Universal Robots PolyScope program: main.urp

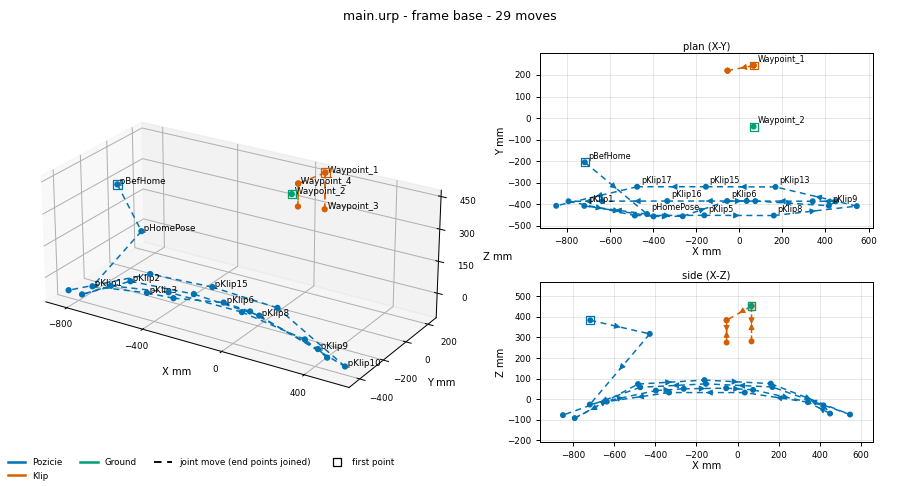
[picture p0: tool path of main.urp in frame base, 29 of 29 moves have a stored position in this frame; points joined in program order, loops and branches not executed]
Program main (installation=default directory=/programs/standart createdIn=5.9.4.1031232 lastSavedIn=3.15.3.106223 robotSerialNumber=2019351917)
Calibrated DH parameters: a=[0.000102, -0.047078, -0.0018, 0.000113, -0.000057, 0]; d=[0.089076, 134.205243, 65.197866, -199.293136, 0.094778, 0.082594]; alpha=[1.569561, -0.003151, -0.001967, 1.571153, -1.570968, 0]; deltaTheta=[0.00002, -1.459967, -0.106279, 1.566186, -0.000048, 0.000035]
Robot Program (runOnlyOnce=false)
  pTarget := p[0,0,0,0,0,0]
  nKlipNo := 1
  SuppressedNode
    bInHome := False
  Script file /programs/standart/loop.script
    | def main():
    | SetMovementsExtParams()
    | while (True):
    |     global niActionNo = read_input_integer_register(2)
    |     sync()
    | 	if (0 == niActionNo):
    | 		sync()
    | 	elif (1 == niActionNo):
    | 		if (read_output_integer_register(2)==255):
    |                                       Klip()
    | 	                  end
    | 	elif (100 == niActionNo):
    | 		if (read_output_integer_register(2)==255):
    | 		Ground()
    | 		end
    | 	elif (254 == niActionNo):
    | 		if (read_output_integer_register(2)==255):
    | 		SetMovementsExtParams ()
    | 		WriteMovementsExtParams ()
    | 		end
    | 	elif (255 == niActionNo):
    | 		sync()
    | 	else:
    | 		popup("nespravne cislo", "Message", False, True, blocking=False)
    | 		halt
    | 	end
    | 	global qActionNumber = niActionNo
    | 	WriteMovementsExtParams ()
    |                   sync()
    | end
    | end
    | def SetMovementsExtParams():
    |     global qActionNumber = read_input_integer_register(2)
    |     global ActGlobalSpeed=read_input_integer_register(3)
    |     global ActualToolNmbr=read_input_integer_register(4)
    |     global ActualWobjNmbr=read_input_integer_register(5)
    |     global ActualPointNmbr=read_input_integer_register(6)
    |     global ActUsrSpecSpd1=read_input_float_register(0)
    |     global ActUsrSpecSpd2=read_input_float_register(1)
    |     global ActCoordX=read_input_float_register(2)
    |     global ActCoordY=read_input_float_register(3)
    |     global ActCoordZ=read_input_float_register(4)
    |     global ActCoordRx=read_input_float_register(5)
    |     global ActCoordRy=read_input_float_register(6)
    |     global ActCoordRz=read_input_float_register(7)
    | end
    | def WriteMovementsExtParams():
    |     write_output_integer_register(2, qActionNumber)
    |     write_output_integer_register(3, ActGlobalSpeed)
    |     write_output_integer_register(4, ActualToolNmbr)
    |     write_output_integer_register(5, ActualWobjNmbr)
    |     write_output_integer_register(6, ActualPointNmbr)
    |     write_output_float_register(0, ActUsrSpecSpd1)
    |     write_output_float_register(1, ActUsrSpecSpd2)
    |     write_output_float_register(2, ActCoordX)
    |     write_output_float_register(3, ActCoordY)
    |     write_output_float_register(4, ActCoordZ)
    |     write_output_float_register(5, ActCoordRx)
    |     write_output_float_register(6, ActCoordRy)
    |     write_output_float_register(7, ActCoordRz)
    | end
  bTest := False
  SuppressedNode
    ipLastPos := get_actual_tcp_pose()
  SuppressedNode
    Call Ground
  Script: main()
SubProgram Pozicie (keepSynchronizedWithDisk=false)
  MoveJ speed 60 deg/s, acceleration 80 deg/s^2 (useActiveTCP=false) tcp=klipBezProtikus
    Waypoint pBefHome: TCP in base x=-715.649 y=-205.001 z=383.699 mm, rx=-2.2037 ry=-0.1236 rz=2.19 rad; joints [-138.345, -84.396, -124.639, -152.449, -62.006, -181.389] deg; flange x=-522.449 y=-193.771 z=341.759 mm, rx=-1.0723 ry=-1.4196 rz=1.3498 rad
    SuppressedNode
      Waypoint Waypoint_46: TCP in base x=-415.026 y=-230.779 z=167.281 mm, rx=-1.4886 ry=-2.6151 rz=0.3802 rad; joints [224.112, -91.25, -119.014, -236.004, -90.455, -253.965] deg; flange x=-396.865 y=-162.684 z=352.334 mm, rx=0.7585 ry=-2.9968 rz=0.0685 rad
    Waypoint pHomePose: motionParameters(blendRadius=0.05); TCP in base x=-426.741 y=-445.009 z=317.531 mm, rx=0.09 ry=-2.3315 rz=2.0367 rad; joints [-141.68, -91.952, -115.104, -182.866, -136.488, -294.8] deg; flange x=-471.084 y=-254.443 z=348.022 mm, rx=1.4686 ry=-1.4379 rz=0.9969 rad
  MoveJ speed 60 deg/s, acceleration 80 deg/s^2 (useActiveTCP=false) tcp=klipProtitlak
    Waypoint pKlip1: motionParameters(jointSpeed=2.094395 jointAcceleration=3.490659 cartesianSpeed=0.25 cartesianAcceleration=1.2); TCP in base x=-717.916 y=-407.007 z=-25.646 mm, rx=-2.1837 ry=2.0431 rz=-0.2819 rad; joints [-139.39, -122.492, -100.341, -46.423, -267.896, -230.294] deg; flange x=-758.162 y=-445.184 z=164.444 mm, rx=3.0989 ry=0.0292 rz=0.0301 rad
    Waypoint pKlip3: TCP in base x=-397.127 y=-455.596 z=42.237 mm, rx=-2.2464 ry=2.1402 rz=-0.0817 rad; joints [-116.855, -94.906, -132.082, -38.147, -277.33, -207.158] deg; flange x=-408.449 y=-427.485 z=238.512 mm, rx=3.1133 ry=0.0064 rz=-0.2302 rad
    Waypoint pKlip4: TCP in base x=-261.696 y=-455.216 z=50.966 mm, rx=-2.2467 ry=2.1402 rz=-0.0816 rad; joints [-102.622, -85.622, -139.646, -41.752, -278.247, -192.808] deg; flange x=-273.005 y=-427.094 z=247.24 mm, rx=3.1132 ry=0.0066 rz=-0.2303 rad
    Waypoint pKlip6: TCP in base x=-55.729 y=-384.407 z=53.915 mm, rx=2.2671 ry=-2.1584 rz=0.0011 rad; joints [-71.993, -75.789, -145.674, -51.415, -282.439, -161.677] deg; flange x=-50.779 y=-426.253 z=247.399 mm, rx=3.1035 ry=0.0081 rz=-0.3413 rad
    Waypoint pKlip7: TCP in base x=74.794 y=-384.809 z=45.787 mm, rx=2.2668 ry=-2.1583 rz=0.0012 rad; joints [-55.209, -77.405, -144.751, -54.17, -281.1, -144.583] deg; flange x=79.767 y=-426.6 z=239.281 mm, rx=3.1032 ry=0.008 rz=-0.3415 rad
    Waypoint pKlip9: TCP in base x=415.982 y=-406.314 z=-29.655 mm, rx=2.0484 ry=-1.9483 rz=-0.4078 rad; joints [-26.071, -109.42, -118.061, -74.534, -286.071, -111.582] deg; flange x=495.201 y=-447.711 z=147.042 mm, rx=2.9746 ry=0.0123 rz=-0.9451 rad
    SuppressedNode
      Waypoint Waypoint_36: TCP in base x=324.659 y=-377.766 z=383.702 mm, rx=-0.149 ry=1.7717 rz=-0.7957 rad; joints [322.849, -58.337, -129.745, -187.968, -109.913, 142.997] deg; flange x=158.512 y=-281.184 z=433.798 mm, rx=-1.7432 ry=1.3314 rz=-1.567 rad
    Waypoint pKlip11: TCP in base x=448.509 y=-385.741 z=-69.2 mm, rx=-2.1761 ry=-2.1899 rz=0.049 rad; joints [-21.41, -106.712, -137.424, -18.115, -266.245, 71.195] deg; flange x=458.564 y=-345.107 z=124.344 mm, rx=0.0574 ry=2.9899 rz=0.0308 rad
    Waypoint pKlip12: TCP in base x=341.02 y=-385.606 z=-13.953 mm, rx=-2.1522 ry=-2.1654 rz=0.1026 rad; joints [-25.586, -93.527, -143.331, -28.169, -266.914, 66.968] deg; flange x=360.406 y=-344.605 z=178.802 mm, rx=0.0584 ry=3.0382 rz=0.027 rad
    Waypoint pKlip14: TCP in base x=34.614 y=-384.474 z=32.579 mm, rx=-2.1881 ry=-2.2026 rz=0.0261 rad; joints [-58.228, -68.011, -154.767, -42.655, -261.175, 34.579] deg; flange x=40.264 y=-343.538 z=226.238 mm, rx=0.0562 ry=2.9672 rz=0.029 rad
    Waypoint pKlip16: TCP in base x=-333.423 y=-384.697 z=32.621 mm, rx=-2.1593 ry=-2.2797 rz=-0.0282 rad; joints [-117.379, -86.002, -139.546, -51.671, -259.578, -28.311] deg; flange x=-339.362 y=-343.904 z=226.302 mm, rx=-0.0144 ry=2.9183 rz=0.037 rad
    Waypoint pKlip18: TCP in base x=-635.307 y=-385.022 z=-11.351 mm, rx=2.0897 ry=2.2082 rz=0.1692 rad; joints [-141.865, -112.773, -110.469, -63.994, -259.039, -53.917] deg; flange x=-667.328 y=-344.256 z=179.762 mm, rx=-0.0161 ry=2.7829 rz=0.0348 rad
    Waypoint pKlip19: TCP in base x=-791.11 y=-385.677 z=-91.337 mm, rx=2.0027 ry=2.1167 rz=0.3408 rad; joints [-149.226, -131.492, -87.605, -78.107, -257.456, -62.68] deg; flange x=-853.946 y=-347.011 z=92.424 mm, rx=-0.0152 ry=2.6186 rz=0.0469 rad
  MoveJ speed 60 deg/s, acceleration 80 deg/s^2 (useActiveTCP=false) tcp=klipBezProtikus
    Waypoint pKlip2: TCP in base x=-483.859 y=-451.884 z=73.894 mm, rx=-2.2466 ry=2.1403 rz=-0.0817 rad; joints [-120.808, -101.736, -119.856, -43.059, -277.036, -211.134] deg; flange x=-492.737 y=-493.65 z=267.254 mm, rx=3.1132 ry=0.0065 rz=-0.2303 rad
    Waypoint pKlip5: TCP in base x=-161.364 y=-450.889 z=93.263 mm, rx=2.2668 ry=-2.1584 rz=0.0013 rad; joints [-87.222, -82.787, -136.209, -50.492, -282.819, -177.268] deg; flange x=-156.42 y=-492.687 z=286.757 mm, rx=3.1033 ry=0.0079 rz=-0.3413 rad
    Waypoint pKlip8: TCP in base x=160.789 y=-451.854 z=75.97 mm, rx=2.2666 ry=-2.1584 rz=0.0036 rad; joints [-51.599, -84.791, -134.791, -57.341, -280.729, -140.913] deg; flange x=165.557 y=-493.433 z=269.515 mm, rx=3.1023 ry=0.0076 rz=-0.3398 rad
    Waypoint pKlip10: TCP in base x=545.477 y=-408.071 z=-73.997 mm, rx=-0.0027 ry=-3.1325 rz=-0.0126 rad; joints [-26.569, -110.661, -126.204, -39.275, -259.338, -24.326] deg; flange x=503.576 y=-410.94 z=119.516 mm, rx=-2.0629 ry=2.1594 rz=0.2484 rad
    Waypoint pKlip13: TCP in base x=168.592 y=-319.265 z=59.545 mm, rx=-2.1886 ry=-2.2026 rz=0.0269 rad; joints [-30.415, -60.616, -155.192, -45.97, -264.32, 62.469] deg; flange x=174.28 y=-278.219 z=253.179 mm, rx=0.0565 ry=2.9673 rz=0.0281 rad
    Waypoint pKlip15: TCP in base x=-154.177 y=-318.207 z=74.988 mm, rx=-2.1599 ry=-2.2798 rz=-0.0278 rad; joints [-93.971, -58.689, -151.594, -62.02, -257.408, -4.458] deg; flange x=-160.141 y=-277.313 z=268.646 mm, rx=-0.014 ry=2.9181 rz=0.0362 rad
    Waypoint pKlip17: TCP in base x=-473.001 y=-318.443 z=58.264 mm, rx=2.0896 ry=2.208 rz=0.1694 rad; joints [-137.201, -93.549, -126.886, -65.846, -257.552, -49.322] deg; flange x=-505.057 y=-277.679 z=249.371 mm, rx=-0.016 ry=2.7827 rz=0.0348 rad
    Waypoint pKlip20: TCP in base x=-848.24 y=-406.643 z=-76.968 mm, rx=3.1026 ry=0.0781 rz=0.1472 rad; joints [-145.711, -128.367, -96.758, -41.883, -255.528, 34.936] deg; flange x=-823.353 y=-396.787 z=119.233 mm, rx=2.0467 ry=2.0412 rz=-0.1418 rad
SubProgram -> Ground
SubProgram Klip (keepSynchronizedWithDisk=false)
  MoveJ speed 60 deg/s, acceleration 80 deg/s^2 (useActiveTCP=true)
    Waypoint Waypoint_1: TCP in base x=67.124 y=243.667 z=452.669 mm, rx=1.0715 ry=1.7614 rz=-1.9585 rad; joints [89.566, -105.051, -69.477, -174.878, 99.822, -221.078] deg; flange x=99.529 y=437.579 z=429.018 mm, rx=0.5733 ry=-1.9692 rz=1.5251 rad
  MoveJ speed 60 deg/s, acceleration 80 deg/s^2 (useActiveTCP=true)
    Waypoint Waypoint_3: TCP in base x=67.172 y=243.612 z=281.105 mm, rx=1.0718 ry=1.7616 rz=-1.9585 rad; joints [89.537, -107.834, -91.269, -150.3, 99.808, -221.132] deg; flange x=99.609 y=437.524 z=257.502 mm, rx=0.5732 ry=-1.9694 rz=1.5248 rad
  Wait Sleep waitTime=1
  MoveJ speed 60 deg/s, acceleration 80 deg/s^2 (useActiveTCP=true)
    Waypoint Waypoint_1: TCP in base x=67.124 y=243.667 z=452.669 mm, rx=1.0715 ry=1.7614 rz=-1.9585 rad; joints [89.566, -105.051, -69.477, -174.878, 99.822, -221.078] deg; flange x=99.529 y=437.579 z=429.018 mm, rx=0.5733 ry=-1.9692 rz=1.5251 rad
  MoveJ speed 60 deg/s, acceleration 80 deg/s^2 (useActiveTCP=true)
    Waypoint Waypoint_4: TCP in base x=-53.847 y=219.832 z=383.966 mm, rx=1.0715 ry=1.7616 rz=-1.9587 rad; joints [103.664, -99.77, -86.087, -162.703, 113.693, -218.301] deg; flange x=-21.424 y=413.743 z=360.331 mm, rx=0.5733 ry=-1.9691 rz=1.5248 rad
  MoveJ speed 60 deg/s, acceleration 80 deg/s^2 (useActiveTCP=true)
    Waypoint Waypoint_5: TCP in base x=-53.781 y=219.797 z=275.539 mm, rx=1.0716 ry=1.7617 rz=-1.9585 rad; joints [103.65, -103.22, -98.22, -147.125, 113.677, -218.327] deg; flange x=-21.362 y=413.713 z=251.934 mm, rx=0.5733 ry=-1.9693 rz=1.5248 rad
  MoveJ speed 60 deg/s, acceleration 80 deg/s^2 (useActiveTCP=true)
    Waypoint Waypoint_4: TCP in base x=-53.847 y=219.832 z=383.966 mm, rx=1.0715 ry=1.7616 rz=-1.9587 rad; joints [103.664, -99.77, -86.087, -162.703, 113.693, -218.301] deg; flange x=-21.424 y=413.743 z=360.331 mm, rx=0.5733 ry=-1.9691 rz=1.5248 rad
Thread Thread_1 (runOnlyOnce=false)
  Script: sync()
  jointPos := get_actual_joint_positions()
SubProgram Ground (keepSynchronizedWithDisk=false)
  Wait Sleep waitTime=2
  MoveJ speed 60 deg/s, acceleration 80 deg/s^2 (useActiveTCP=true)
    Waypoint Waypoint_2: TCP in base x=67.125 y=-39.539 z=452.728 mm, rx=1.0717 ry=1.7615 rz=-1.9585 rad; joints [88.851, -66.59, -104.923, -177.907, 99.247, -221.206] deg; flange x=99.558 y=154.372 z=429.109 mm, rx=0.5732 ry=-1.9693 rz=1.5249 rad
